Yaskawa INFORM job: X2_50&56A(90,0).JBI

/JOB
//NAME X2_50&56A(90,0)
//POS
///NPOS 396,396,396,18,0,0
///TOOL 0
///POSTYPE PULSE
///PULSE
C00000=35013,-75230,-81678,29902,96544,-59223
C00001=35013,-75230,-81678,29902,96544,50582
C00002=120856,-140422,-87858,-20775,49685,84873
C00003=94802,-63197,-51322,-24283,84063,77554
C00004=130027,34169,-1600,32218,111617,-60978
C00005=146238,55672,63206,30358,82483,-64229
C00006=147931,55156,65583,30589,80380,-64138
C00007=88821,-39952,-28103,-20433,93116,74064
C00008=88821,-39522,-26790,-20414,92564,74158
C00009=88821,-39864,-27834,-20427,93002,74084
C00010=88103,-42626,-29535,-20492,92474,73914
C00011=88821,-39864,-27834,-20427,93002,74084
C00012=78489,-20820,-14449,-12623,103903,88788
C00013=79217,-21691,-15077,-12445,103957,89045
C00014=78489,-21142,-15590,-12658,104428,88732
C00015=86357,-31648,-34432,-18066,105893,79829
C00016=106408,-49809,-40215,-13540,104251,87431
C00017=105408,-58256,-44905,-13671,102667,87249
C00018=105408,-58256,-44905,-13671,102667,87249
C00019=110503,10444,25613,-12126,95572,-74078
C00020=112000,-36737,-25207,-22040,88152,-84766
C00021=112000,-31881,-11932,-22145,82876,-83796
C00022=112000,-30399,-8347,-22203,81533,-83546
C00023=112000,-31881,-11932,-22145,82876,-83796
C00024=116556,-31988,-11028,-21876,83512,-82269
C00025=116556,-30496,-7483,-21927,82195,-82028
C00026=116476,-32903,-9067,-21944,81929,-82006
C00027=116556,-30496,-7483,-21927,82195,-82028
C00028=116556,-30496,-7483,-21927,82195,-82028
C00029=115731,-30414,-7427,-21987,81986,-82285
C00030=116556,-30496,-7483,-21927,82195,-82028
C00031=106621,-34317,-21280,-11409,87224,-86882
C00032=68546,9416,10683,-17932,104217,-63227
C00033=68516,6763,11888,-17759,102202,-62934
C00034=69948,4612,13298,-17270,100624,-62182
C00035=69948,5621,16125,-17192,99456,-62015
C00036=69948,5087,14650,-17232,100063,-62102
C00037=67463,10522,20606,-17770,98699,-62796
C00038=66929,8958,19215,-17898,98632,-62977
C00039=67463,10522,20606,-17770,98699,-62796
C00040=68831,9536,19728,-17449,99024,-62352
C00041=69409,8421,18742,-17312,99180,-62168
C00042=68137,9624,17362,-17710,100309,-62790
C00043=69946,10003,12499,-17525,103743,-62639
C00044=115698,-30544,-51433,-15731,84190,-63390
C00045=118338,-32636,-46922,-7735,73478,-10834
C00046=113479,46792,28572,-8285,94763,37933
C00047=101095,55404,42650,-8147,89306,34054
C00048=100229,58556,52121,-8145,85049,34033
C00049=99767,59813,55030,-8149,83870,33952
C00050=99764,60521,57124,-8160,82954,34012
C00051=99767,59813,55030,-8149,83870,33952
C00052=102778,57366,53086,-13194,83019,35153
C00053=102079,58061,53874,-13178,82781,34934
C00054=102778,57366,53086,-13194,83019,35153
C00055=103317,56175,50346,-13188,84155,35220
C00056=104672,52489,39292,-13191,89159,35160
C00057=104701,56902,48819,-15320,94256,69233
C00058=104701,57353,50315,-15300,93589,69317
C00059=104701,57270,50045,-15303,93709,69302
C00060=104511,53820,46175,-15336,94260,69166
C00061=104638,55892,48016,-15323,94215,69218
C00062=105717,54144,46059,-15234,94714,69537
C00063=105635,50040,42095,-15252,95019,69470
C00064=105236,50331,42415,-15286,94898,69344
C00065=105635,49167,38717,-15311,96595,69274
C00066=102055,-19938,-28050,-3892,79498,23263
C00067=101482,-35884,-39735,-11033,71484,5125
C00068=99031,-31158,-27485,-14483,64579,4851
C00069=99281,-29511,-26374,-14550,64779,4920
C00070=99247,-29735,-26526,-14541,64752,4910
C00071=99247,-29464,-25406,-14605,64218,4980
C00072=99051,-31169,-27981,-14456,64871,4820
C00073=96268,-39480,-34083,-4840,61268,-4619
C00074=96136,-35876,-28725,-4851,59820,-4606
C00075=95241,-35325,-28368,-4481,59831,-4954
C00076=96136,-35958,-29023,-4844,59961,-4612
C00077=124050,-15750,-20412,-8746,80746,42462
C00078=136003,-35750,-34405,-10595,80538,46616
C00079=134863,-34094,-26254,-10570,76291,46583
C00080=136016,-32722,-22756,-10798,75019,47102
C00081=136016,-31890,-20154,-10854,73866,47205
C00082=136016,-32408,-21756,-10817,74572,47142
C00083=116377,-35025,-23683,16914,73563,39729
C00084=116394,-34210,-21577,16985,72720,39615
C00085=115269,-34083,-21492,17148,72970,39239
C00086=117663,-35285,-24614,16688,73723,40220
C00087=141315,-33561,-31051,-11181,80302,48491
C00088=136363,-34899,-19347,-7835,84694,46414
C00089=120104,-33911,-11600,-8301,78857,41249
C00090=118071,-31578,-6204,-8386,76551,40710
C00091=117257,-30555,-3964,-8424,75624,40496
C00092=117257,-29687,-2023,-8450,74882,40547
C00093=117257,-30555,-3964,-8424,75624,40496
C00094=122539,-29708,-1883,-13613,75634,42844
C00095=121317,-29732,-1900,-13643,75432,42443
C00096=122539,-29708,-1883,-13613,75634,42844
C00097=123471,-30618,-3978,-13546,76585,43059
C00098=125796,-32661,-9010,-13387,78955,43601
C00099=120122,-41338,-8990,-8476,73493,41622
C00100=117871,-38446,-3197,-8601,71207,41016
C00101=116972,-37197,-791,-8654,70286,40775
C00102=116972,-36136,1298,-8692,69554,40829
C00103=116972,-37197,-791,-8654,70286,40775
C00104=122649,-36403,912,-13956,70634,43458
C00105=121298,-36427,896,-13995,70410,43017
C00106=122649,-36403,912,-13956,70634,43458
C00107=120043,-14467,15179,-12402,85308,69300
C00108=120029,-16401,14941,-12417,84477,69377
C00109=120021,-18007,13765,-12421,84376,69384
C00110=120029,-16401,14941,-12417,84477,69377
C00111=123681,-37514,-1336,-13860,71590,43701
C00112=126252,-40055,-6735,-13636,73968,44314
C00113=154326,-120554,-77654,-11334,79888,63138
C00114=167720,-105639,-119673,-16034,110248,69380
C00115=180425,17295,-38776,-18903,121217,77748
C00116=161552,-71669,-79142,-10296,105844,81662
C00117=160864,-75997,-77577,-10180,102620,81695
C00118=159718,-74822,-75193,-10227,101627,81377
C00119=159595,-74270,-73499,-10203,100862,81396
C00120=160050,-75992,-74945,-10170,100925,81551
C00121=160240,-80173,-76229,-10103,99611,81726
C00122=160318,-76812,-75188,-10139,100690,81664
C00123=161300,-71121,-77557,-10275,105130,81635
C00124=122590,-90956,-95479,6285,107811,74232
C00125=122432,-96187,-93928,6136,104200,73988
C00126=122366,-98076,-93201,6086,102795,73894
C00127=122349,-96392,-90986,6070,102302,73864
C00128=122333,-96702,-91360,6071,102373,73862
C00129=121172,-100063,-92157,5915,101229,73400
C00130=122333,-96702,-91360,6071,102373,73862
C00131=116908,-96303,-91435,5489,103011,71994
C00132=118888,-98383,-91954,5688,102128,72646
C00133=116908,-96303,-91435,5489,103011,71994
C00134=117392,-89431,-93773,5700,107925,72394
C00135=123779,-92334,-96085,-11860,100478,68930
C00136=121799,-96099,-93963,-11739,97018,68578
C00137=120978,-97397,-93019,-11702,95677,68421
C00138=120976,-95732,-90808,-11689,95182,68467
C00139=121047,-96000,-91535,-11697,95495,68462
C00140=119860,-99344,-92335,-11668,94123,68181
C00141=121047,-96000,-91535,-11697,95495,68462
C00142=119543,-98346,-92112,-11677,94445,68041
C00143=121592,-100306,-92571,-11657,94029,68789
C00144=119543,-98346,-92112,-11677,94445,68041
C00145=122418,-93690,-95360,-11815,99162,68586
C00146=124052,-92327,-98574,-11935,102020,68874
C00147=122075,-96496,-96608,-11789,98453,68536
C00148=121256,-97943,-95721,-11744,97072,68385
C00149=121250,-96320,-93531,-11728,96567,68431
C00150=121163,-96877,-94234,-11732,96698,68388
C00151=119974,-100369,-95083,-11696,95280,68111
C00152=121163,-96877,-94234,-11732,96698,68388
C00153=120506,-98881,-94746,-11711,95903,68236
C00154=118500,-96784,-94222,-11730,96355,67499
C00155=120506,-98881,-94746,-11711,95903,68236
C00156=123349,-93657,-97773,-11879,100767,68753
C00157=136369,-86264,-75827,-53025,86694,81775
C00158=132228,-88122,-74116,-52932,83075,81639
C00159=130522,-88702,-73354,-52914,81621,81560
C00160=129603,-91514,-73993,-52982,80442,81751
C00161=133099,-92681,-76573,-53031,83062,82125
C00162=131615,-95137,-76568,-53090,81428,82278
C00163=130003,-92998,-74814,-53028,80513,81930
C00164=131615,-95137,-76568,-53090,81428,82278
C00165=125724,-93998,-78752,-52538,79248,80319
C00166=127169,-93644,-77288,-52734,79625,80891
C00167=125724,-93998,-78752,-52538,79248,80319
C00168=131917,-91951,-81421,-52749,84465,80650
C00169=125882,-96985,-97972,-20817,92084,56602
C00170=122325,-98161,-95172,-20440,89016,55857
C00171=120880,-94284,-92066,-20293,88735,55390
C00172=120880,-94153,-90803,-20292,88068,55501
C00173=120880,-94284,-92066,-20293,88735,55390
C00174=119026,-94251,-92054,-20095,88291,54803
C00175=120880,-94284,-92066,-20293,88735,55390
C00176=120884,-98206,-92897,-20294,87320,55628
C00177=120880,-94284,-92066,-20293,88735,55390
C00178=125854,-95536,-95978,-20803,91624,56671
C00179=125850,-66912,-79659,-30836,57983,58657
C00180=122561,-63207,-75462,-29110,56252,57732
C00181=121295,-61670,-73737,-28426,55590,57365
C00182=121291,-60661,-71640,-28674,54906,57565
C00183=121285,-60765,-71809,-28654,54949,57550
C00184=119473,-60737,-71796,-27523,54360,56906
C00185=121285,-60765,-71809,-28654,54949,57550
C00186=119935,-60692,-71734,-27818,54496,57075
C00187=119959,-57359,-70502,-27528,55354,56840
C00188=119935,-60692,-71734,-27818,54496,57075
C00189=124401,-66105,-77764,-30230,56821,58377
C00190=128142,-64639,-90036,-18676,74706,62694
C00191=138485,-71827,-101197,11106,105399,77644
C00192=147024,-87385,-83593,35439,109592,87133
C00193=149732,-92665,-83137,35225,106008,87097
C00194=151109,-95679,-83834,35232,104517,87192
C00195=150643,-92710,-80195,35037,104118,86860
C00196=144971,-96193,-77741,39215,100748,74661
C00197=143884,-94649,-78323,39224,102144,74704
C00198=141496,-90316,-79520,39399,105550,74933
C00199=154875,-73459,-94031,-3699,115712,75473
C00200=154642,-88430,-80864,-46638,100530,71967
C00201=150685,-92332,-80273,-46535,96810,71811
C00202=149068,-93915,-80023,-46523,95290,71747
C00203=152233,-91403,-76041,-46197,96115,72893
C00204=138023,-100193,-87798,-32403,89280,71025
C00205=139486,-99224,-88637,-32451,90704,71199
C00206=143008,-96307,-90518,-32622,94313,71562
C00207=126401,-92982,-99947,-26116,71912,46119
C00208=122401,-89174,-95921,-24616,70248,44972
C00209=121170,-87691,-94393,-24143,69731,44617
C00210=121073,-40431,-77118,-23973,104037,41292
C00211=121948,-141376,-105315,-24084,72465,47862
C00212=119793,-124223,-100539,-21665,86903,40754
C00213=121070,-126388,-102412,-21638,87354,41108
C00214=126026,-127807,-105919,-21532,89991,42436
C00215=136654,-67846,-101646,5444,103045,74682
C00216=128322,-96725,-99076,-14451,99613,67284
C00217=128011,-95143,-96681,-14417,98917,67259
C00218=125059,-98267,-95078,-14269,95825,66574
C00219=132883,-103944,-96240,-14189,95056,69399
C00220=122114,-97273,-96139,-7492,99903,69823
C00221=123656,-92823,-98050,-7552,103478,70135
C00222=148370,-106244,-91268,-32547,97235,62203
C00223=143957,-109023,-89633,-32719,93465,61524
C00224=142187,-110300,-89017,-32799,91899,61269
C00225=110014,-102343,-95219,-10833,94604,66470
C00226=122878,-112804,-97097,-10537,93258,71032
C00227=110561,-104342,-93907,-1603,99479,78541
C00228=110841,-84726,-85708,-1760,111290,78449
C00229=111201,-78802,-86432,-1737,114786,78527
C00230=107617,-60482,-79878,-8180,107350,64339
C00231=106036,-64346,-78204,-8057,104211,64009
C00232=105256,-65205,-77316,-8026,103160,63809
C00233=107559,-69233,-78771,-7955,102216,64664
C00234=165613,-100062,-83585,-4761,94184,85074
C00235=168997,-99278,-82863,-4484,94340,86226
C00236=170567,-98725,-82495,-4354,94483,86758
C00237=166939,-94886,-91891,-4771,102005,85231
C00238=180121,-120623,-113011,-11864,94268,89792
C00239=202989,-63880,-99903,-47799,99542,84030
C00240=168472,-147890,-132681,-14947,97151,71352
C00241=154326,-120554,-77654,-11334,79888,63138
C00242=128098,-77833,-51544,1657,63239,16727
C00243=116532,-49017,-34945,4360,90951,81305
C00244=116532,-49017,-34945,4360,90951,81305
C00245=116798,-50663,-32111,4378,88355,81305
C00246=118979,-64696,-37015,4666,76602,81617
C00247=127924,-64268,-36804,4494,76190,84659
C00248=124228,-50732,-32149,5002,87911,83800
C00249=145745,-14259,570,-10366,107018,74117
C00250=151803,-16835,2182,-12669,103763,71943
C00251=152120,-15652,4819,-12499,102817,72155
C00252=153130,-16591,-3293,-13485,106909,71001
C00253=99208,-22167,-7317,16130,105202,90552
C00254=102975,-22456,-1750,16076,101623,90323
C00255=102764,-21603,-119,15971,101119,90180
C00256=102764,-21410,336,15959,100945,90157
C00257=100868,-20755,-6903,14931,106373,89315
C00258=123764,-49143,-35016,4968,90511,83746
C00259=123498,-46334,-32145,-14225,106729,81506
C00260=122671,-49917,-31274,-14287,104276,81501
C00261=124642,-51419,-28814,-13533,102390,82429
C00262=121239,-51674,-29154,-14566,101882,81278
C00263=121239,-51674,-29154,-14566,101882,81278
C00264=121239,-51674,-29154,-14566,101882,81278
C00265=119414,-50002,-31488,-15265,103772,80384
C00266=116044,-49795,-31370,-16241,103155,79243
C00267=108003,-52785,-29324,-8850,97765,81124
C00268=118660,-64605,-35307,-15810,90578,70895
C00269=127566,-70492,-45301,-19994,92283,73343
C00270=120368,-46468,-32388,-15179,106240,80415
C00271=103583,-18395,-21065,-18333,98049,47386
C00272=95522,-2033,346,-19157,86542,33647
C00273=95065,-1179,4289,-19188,84551,33796
C00274=94955,-858,5669,-19196,83900,33869
C00275=92999,-12490,-3621,-19193,83196,33279
C00276=91633,5412,10982,-17435,91860,45178
C00277=96102,40486,49560,-22978,105705,40202
C00278=95175,38955,47637,-23356,105815,39825
C00279=95175,41860,54365,-23036,103374,40320
C00280=96604,40287,46680,-23025,107388,40051
C00281=97434,43818,44752,-23189,110389,39758
C00282=95302,21282,15864,-17128,100326,40606
C00283=95633,-1961,-1285,-16168,78923,31701
C00284=94125,315,3726,-16087,76781,31446
C00285=94086,2267,8889,-16221,74681,31714
C00286=93769,3603,11937,-16272,73472,31765
C00287=95210,13761,20912,-16469,73473,32289
C00288=95827,11154,15194,-16384,75690,32206
C00289=95302,10808,12912,-16245,76762,31872
C00290=94760,268,4885,-16208,76196,31753
C00291=94118,1970,8158,-16204,74972,31685
C00292=93771,3565,12382,-16293,73191,31803
C00293=95246,13304,20868,-16485,73277,32327
C00294=95842,10702,14076,-16353,76128,32151
C00295=96013,9170,10401,-16290,77582,32017
C00296=97216,11756,13085,-16445,77515,32459
C00297=97106,13151,16539,-16517,76140,32606
C00298=96699,14660,19946,-16558,74788,32646
C00299=97321,19796,24727,-16651,74625,32895
C00300=91528,6104,12814,-7587,65442,17765
C00301=89231,-9641,862,-3829,57239,21101
C00302=86569,-23656,-15616,-815,55978,22098
C00303=99387,-43194,-40222,-6284,61646,26942
C00304=121163,28995,9538,-19255,89803,33709
C00305=111536,74157,50908,-19383,94154,29578
C00306=110126,77328,60869,-19265,89563,29800
C00307=109597,77904,61840,-18115,89315,29667
C00308=107134,62574,43702,-13173,82287,21832
C00309=105849,37660,21975,-10686,72529,22941
C00310=108144,30390,14425,-11303,73735,23647
C00311=110038,48233,28322,-17563,85893,26316
C00312=110492,45790,38116,-18907,91301,38258
C00313=109482,39772,34705,-18931,90124,38079
C00314=108901,41209,40132,-18939,87523,38277
C00315=108525,40703,40973,-18962,86700,38272
C00316=107041,55931,58526,-17360,94880,40074
C00317=107089,67852,69975,-15460,97104,40498
C00318=107063,68178,67130,-13775,98442,40242
C00319=113418,36081,17598,-23566,90539,39080
C00320=113418,36081,17598,-23168,95829,82784
C00321=113828,51923,41074,-24171,98232,82423
C00322=112579,52431,41633,-24296,97790,82045
C00323=112126,56349,44369,-24366,97957,81836
C00324=108217,58430,46714,-24702,96454,80681
C00325=108494,54192,43684,-24661,96249,80828
C00326=108007,54490,44017,-24701,96056,80686
C00327=107594,60273,47410,-24788,96737,80387
C00328=114507,54753,41023,-24220,99790,82353
C00329=122054,71046,63948,-32664,112221,61348
C00330=123579,46190,40204,-38346,104555,54529
C00331=124736,37096,33930,-39238,101677,53630
C00332=124818,38918,39542,-38856,99735,54394
C00333=126462,40069,35828,-39705,101719,52991
C00334=128176,30389,18653,-40526,106846,51750
C00335=130467,-19777,-28453,-43779,86857,-28489
C00336=121945,-40313,-29836,-49261,62361,-22447
C00337=123791,-37570,-24592,-50353,62174,-21277
C00338=114538,-37294,-24521,-48212,57212,-23703
C00339=116456,-42529,-32983,-47605,59952,-24171
C00340=113288,-38496,-19602,-52049,50370,-20126
C00341=111978,-38266,-19460,-51659,49655,-20498
C00342=111880,-40713,-23013,-51024,50195,-20951
C00343=122010,-41537,-23518,-53640,55853,-18263
C00344=118733,-42874,-23495,-50076,50608,-22105
C00345=115692,-42672,-23415,-49110,48994,-23003
C00346=119979,-48793,-33564,-48599,53387,-23123
C00347=127641,-44516,-39522,-49206,67999,-22470
C00348=137272,-90960,-86846,-29989,75596,51153
C00349=137772,-94948,-88443,-30238,74846,51554
C00350=80124,-23753,-1605,24425,88616,-57626
C00351=97606,38320,19913,32229,69524,-73177
C00352=104908,49911,44038,31966,59160,-73213
C00353=105731,66374,62732,32681,56250,-73801
C00354=101009,56188,45401,32602,62685,-73830
C00355=95324,41633,28025,33647,67650,-74589
C00356=87558,19072,373,28757,109210,-81139
C00357=99257,11218,8118,26405,109034,-79116
C00358=100705,8698,11538,26232,105511,-79373
C00359=103992,6523,9295,19718,103157,-78424
C00360=103706,6801,9674,20068,103243,-78529
C00361=103706,6801,9674,20068,103243,-78529
C00362=103175,12796,9745,21520,108066,-80350
C00363=94457,17964,8722,13249,111502,-83272
C00364=77268,-3254,-24039,37164,82398,-77433
C00365=55933,-99496,-79908,41589,80337,-87481
C00366=92475,-142040,-80472,-3538,45591,39607
C00367=111759,-138997,-77779,-20724,42469,82604
C00368=123409,-124840,-68778,-23994,47004,86899
C00369=115111,-123372,-67292,-17121,44583,82853
C00370=106159,-121342,-66429,-9144,43886,78109
C00371=56877,-95499,-59936,14598,58195,57192
C00372=67543,-97387,-64583,11943,58838,61427
C00373=85335,-36233,-33573,-15386,101650,67363
C00374=22776,-147712,-91578,22852,59519,43831
C00375=66236,-86626,-72800,11302,69406,62015
C00376=122101,-60707,-49124,40437,82186,-58582
C00377=76878,-31978,-23741,-7994,99594,69431
C00378=79357,-35161,-25830,-10416,97591,64533
C00379=82324,-46618,-32975,-14804,90128,52114
C00380=86643,-46469,-34772,-14478,92051,53396
C00381=73286,-4461,-1127,-6755,115907,88976
C00382=73225,-6334,-1269,-6726,115035,89004
C00383=71733,-2264,5245,-7236,112998,88564
C00384=76479,-5255,-4471,-10939,116481,85182
C00385=98335,-62985,-54253,-3239,96100,60563
C00386=98335,-62985,-54253,-3239,96100,60563
C00387=98335,-62985,-54253,-3239,96100,60563
C00388=152493,16707,-760,-6447,101329,44907
C00389=169300,37694,50213,-44743,100506,44736
C00390=167112,29738,44456,-45250,99025,44384
C00391=162955,52490,68578,-45996,94710,44438
C00392=158969,29363,17393,-36895,102134,39004
C00393=132653,-84295,-81500,4027,86761,-71858
C00394=118286,-84176,-81449,4028,86790,-71859
C00395=-2286,-108146,-98365,80,72600,-100
BC00000=231000,517456,593434
BC00001=34376,517456,225147
BC00002=102572,425363,301105
BC00003=102572,425363,301105
BC00004=334489,491452,488918
BC00005=322698,517456,378589
BC00006=322698,517456,378589
BC00007=102572,425363,301105
BC00008=102572,425363,301105
BC00009=102572,425363,301105
BC00010=102572,425363,301105
BC00011=102572,425363,301105
BC00012=102572,425363,301105
BC00013=102572,425363,301105
BC00014=102572,425363,301105
BC00015=102572,425363,301105
BC00016=102572,425363,301105
BC00017=102572,579800,381307
BC00018=306896,476295,640078
BC00019=306896,448601,572655
BC00020=271432,459376,401351
BC00021=271432,459376,401351
BC00022=271432,459376,401351
BC00023=271432,459376,401351
BC00024=271432,459376,401351
BC00025=271432,459376,401351
BC00026=271432,459376,401351
BC00027=271432,459376,401351
BC00028=271432,459376,401351
BC00029=271432,459376,401351
BC00030=271432,459376,401351
BC00031=271432,459376,401351
BC00032=268738,434477,371771
BC00033=268738,434477,371771
BC00034=268738,434477,371771
BC00035=268738,434477,371771
BC00036=268738,434477,371771
BC00037=268738,434477,371771
BC00038=268738,434477,371771
BC00039=268738,434477,371771
BC00040=268738,434477,371771
BC00041=268738,434477,371771
BC00042=268738,434477,371771
BC00043=268738,434477,371771
BC00044=294080,442709,254978
BC00045=331538,416726,228027
BC00046=305027,399020,290854
BC00047=305027,399020,290854
BC00048=305027,399020,290854
BC00049=305027,399020,290854
BC00050=305027,399020,290854
BC00051=305027,399020,290854
BC00052=305027,399020,290854
BC00053=305027,399020,290854
BC00054=305027,399020,290854
BC00055=305027,399020,290854
BC00056=305027,399020,290854
BC00057=305029,399021,290852
BC00058=305029,399021,290852
BC00059=305029,399021,290852
BC00060=305029,399021,290852
BC00061=305029,399021,290852
BC00062=305029,399021,290852
BC00063=305029,399021,290852
BC00064=305029,399021,290852
BC00065=305029,399021,290852
BC00066=305029,399021,290852
BC00067=305029,399021,290852
BC00068=305029,399021,290852
BC00069=305029,399021,290852
BC00070=305029,399021,290852
BC00071=305029,399021,290852
BC00072=305029,399021,290852
BC00073=305029,399021,290852
BC00074=305029,399021,290852
BC00075=305029,399021,290852
BC00076=305029,399021,290852
BC00077=334039,399020,360133
BC00078=334039,399020,360133
BC00079=334039,399020,360133
BC00080=334039,399020,360133
BC00081=334039,399020,360133
BC00082=334039,399020,360133
BC00083=334039,399020,360133
BC00084=334039,399020,360133
BC00085=334039,399020,360133
BC00086=334039,399020,360133
BC00087=334039,399020,360133
BC00088=367859,399020,440892
BC00089=367859,399020,440892
BC00090=367859,399020,440892
BC00091=367859,399020,440892
BC00092=367859,399020,440892
BC00093=367859,399020,440892
BC00094=367859,399020,440892
BC00095=367859,399020,440892
BC00096=367859,399020,440892
BC00097=367859,399020,440892
BC00098=367859,399020,440892
BC00099=367957,451741,487073
BC00100=367957,451741,487073
BC00101=367957,451741,487073
BC00102=367957,451741,487073
BC00103=367957,451741,487073
BC00104=367957,451741,487073
BC00105=367957,451741,487073
BC00106=367957,451741,487073
BC00107=367957,451741,487073
BC00108=367957,451741,487073
BC00109=367957,451741,487073
BC00110=367957,451741,487073
BC00111=367957,451741,487073
BC00112=367957,451741,487073
BC00113=242061,521422,834580
BC00114=140834,449782,1062640
BC00115=97513,455583,1075193
BC00116=1592,411167,1075139
BC00117=1592,411167,1075139
BC00118=1592,409938,1075139
BC00119=1592,409938,1075139
BC00120=1592,409938,1075139
BC00121=1592,409938,1075139
BC00122=1592,409938,1075139
BC00123=1592,409938,1075139
BC00124=50980,356914,1075139
BC00125=50980,356914,1075139
BC00126=50980,356914,1075139
BC00127=50980,356914,1075139
BC00128=50980,356914,1075139
BC00129=50980,356914,1075139
BC00130=50980,356914,1075139
BC00131=50980,356914,1075139
BC00132=50980,356914,1075139
BC00133=50980,356914,1075139
BC00134=50980,356914,1075139
BC00135=20406,370413,1075139
BC00136=20406,370413,1075139
BC00137=20406,370413,1075139
BC00138=20406,370413,1075139
BC00139=20406,370413,1075139
BC00140=20406,370413,1075139
BC00141=20406,370413,1075139
BC00142=20406,370413,1075139
BC00143=20406,370413,1075139
BC00144=20406,370413,1075139
BC00145=20406,370413,1075139
BC00146=44109,357401,1075139
BC00147=44109,357401,1075139
BC00148=44109,357401,1075139
BC00149=44109,357401,1075139
BC00150=44109,357401,1075139
BC00151=44109,357401,1075139
BC00152=44109,357401,1075139
BC00153=44109,357401,1075139
BC00154=44109,357401,1075139
BC00155=44109,357401,1075139
BC00156=44109,357401,1075139
BC00157=1592,378501,1075139
BC00158=1592,378501,1075139
BC00159=1592,378501,1075139
BC00160=1592,378501,1075139
BC00161=1592,378501,1075139
BC00162=1592,378501,1075139
BC00163=1592,378501,1075139
BC00164=1592,378501,1075139
BC00165=1592,378501,1075139
BC00166=1592,378501,1075139
BC00167=1592,378501,1075139
BC00168=1592,378501,1075139
BC00169=34924,366834,1075139
BC00170=34924,366834,1075139
BC00171=34924,366834,1075139
BC00172=34924,366834,1075139
BC00173=34924,366834,1075139
BC00174=34924,366834,1075139
BC00175=34924,366834,1075139
BC00176=34924,366834,1075139
BC00177=34924,366834,1075139
BC00178=34924,366834,1075139
BC00179=29635,379683,1075139
BC00180=29635,379683,1075139
BC00181=29635,379683,1075139
BC00182=29635,379683,1075139
BC00183=29635,379683,1075139
BC00184=29635,379683,1075139
BC00185=29635,379683,1075139
BC00186=29635,379683,1075139
BC00187=29635,379683,1075139
BC00188=29635,379683,1075139
BC00189=29635,379683,1075139
BC00190=45948,369971,1075139
BC00191=91010,343142,1075139
BC00192=128368,320900,1075139
BC00193=128368,320900,1075139
BC00194=128368,320900,1075139
BC00195=128368,320900,1075139
BC00196=128368,320900,1075139
BC00197=128368,320900,1075139
BC00198=128368,320900,1075139
BC00199=82932,344066,1075139
BC00200=34742,368635,1075139
BC00201=34742,368635,1075139
BC00202=34742,368635,1075139
BC00203=34742,368635,1075139
BC00204=34742,368635,1075139
BC00205=34742,368635,1075139
BC00206=34742,368635,1075139
BC00207=32385,335579,1075139
BC00208=32385,335579,1075139
BC00209=32385,335579,1075139
BC00210=32385,335579,1075139
BC00211=32385,335579,1075139
BC00212=32385,335579,1075139
BC00213=32385,335579,1075139
BC00214=32385,335579,1075139
BC00215=83004,347908,1075139
BC00216=56012,350823,1075139
BC00217=56012,350823,1075139
BC00218=56012,350822,1075135
BC00219=56012,350822,1075135
BC00220=56012,350823,1075139
BC00221=56012,350823,1075139
BC00222=32229,352573,1075139
BC00223=32229,352573,1075139
BC00224=32229,352573,1075139
BC00225=32229,352573,1075139
BC00226=32229,352573,1075139
BC00227=32229,352573,1075139
BC00228=32229,352573,1075139
BC00229=32229,352573,1075139
BC00230=1592,390224,1075139
BC00231=1592,390224,1075139
BC00232=1592,390224,1075139
BC00233=1592,390224,1075139
BC00234=1592,390224,1075139
BC00235=1592,390224,1075139
BC00236=1592,390224,1075139
BC00237=1592,390224,1075139
BC00238=1592,390224,1075139
BC00239=97513,454354,1075193
BC00240=140834,448553,1062640
BC00241=242061,520193,834580
BC00242=311361,456270,477376
BC00243=342823,443238,375594
BC00244=342823,443238,375594
BC00245=342823,443238,375594
BC00246=342823,443238,375594
BC00247=342823,443238,375594
BC00248=342823,443238,375594
BC00249=342823,443238,375594
BC00250=342823,443238,375594
BC00251=342823,443238,375594
BC00252=342823,443238,375594
BC00253=342823,443238,375594
BC00254=342823,443238,375594
BC00255=342823,443238,375594
BC00256=342823,443238,375594
BC00257=342823,443238,375594
BC00258=342823,443238,375594
BC00259=362743,414004,329031
BC00260=362743,414004,329031
BC00261=362743,414004,329031
BC00262=362743,414004,329031
BC00263=362743,414004,329031
BC00264=362743,414004,329031
BC00265=362743,414004,329031
BC00266=362743,414004,329031
BC00267=362743,414004,329031
BC00268=362743,414004,329031
BC00269=362743,414004,329031
BC00270=362743,414004,329031
BC00271=315566,460561,335729
BC00272=294603,481248,338705
BC00273=294603,481248,338705
BC00274=294603,481247,338705
BC00275=294603,481247,338705
BC00276=294603,481247,338705
BC00277=294603,481248,338705
BC00278=294603,481248,338705
BC00279=294603,481248,338705
BC00280=294603,481248,338705
BC00281=294603,481248,338705
BC00282=294603,481248,338705
BC00283=290459,488683,355824
BC00284=290459,488683,355824
BC00285=290459,488683,355824
BC00286=290459,488683,355824
BC00287=290459,488683,355824
BC00288=290459,488683,355824
BC00289=290459,488683,355824
BC00290=290354,460436,354488
BC00291=290354,460436,354488
BC00292=290354,460436,354488
BC00293=290354,460436,354488
BC00294=290354,460436,354488
BC00295=290354,460436,354488
BC00296=293273,446294,341840
BC00297=293273,446294,341840
BC00298=293273,446294,341840
BC00299=293273,446294,341840
BC00300=293273,446294,341840
BC00301=293273,446294,341840
BC00302=293273,446294,341840
BC00303=293273,446294,341840
BC00304=316572,397791,307269
BC00305=317775,402370,174220
BC00306=317775,402370,174220
BC00307=317775,402370,174220
BC00308=317775,402370,174220
BC00309=317775,402370,219932
BC00310=317775,402370,258168
BC00311=317775,402370,227987
BC00312=319614,400694,306223
BC00313=319614,400694,306223
BC00314=319614,400694,306223
BC00315=319614,400694,306223
BC00316=319614,400694,306223
BC00317=319614,400694,306223
BC00318=319614,400694,306223
BC00319=319614,400694,252456
BC00320=319614,400694,252456
BC00321=319614,400694,252456
BC00322=319614,400694,252456
BC00323=319614,400694,252456
BC00324=319614,400694,252456
BC00325=319614,400694,252456
BC00326=319614,400694,252456
BC00327=319614,400694,252456
BC00328=319614,400694,252456
BC00329=319614,400694,252456
BC00330=319614,400694,252456
BC00331=319610,400694,252455
BC00332=319610,400694,252455
BC00333=319614,400694,252456
BC00334=319614,400694,252456
BC00335=319614,400694,252456
BC00336=319614,400694,252456
BC00337=319614,400694,252456
BC00338=319614,400694,252456
BC00339=319614,400694,252456
BC00340=319614,400694,252456
BC00341=319614,400694,252456
BC00342=319614,400694,252456
BC00343=319614,400694,252456
BC00344=319614,400694,252456
BC00345=319614,400694,252456
BC00346=319614,400694,252456
BC00347=319614,400694,252456
BC00348=319614,400694,392080
BC00349=319614,552522,392080
BC00350=396313,516601,467973
BC00351=396313,490351,238820
BC00352=396313,490351,238820
BC00353=396313,490351,238820
BC00354=396313,490351,238820
BC00355=395126,490351,305637
BC00356=395126,490351,305637
BC00357=395126,490351,305637
BC00358=395126,490351,305637
BC00359=395126,490351,305637
BC00360=395126,490351,305637
BC00361=395126,490351,305637
BC00362=395126,490351,305637
BC00363=395126,490351,305637
BC00364=391357,490351,517866
BC00365=391357,520423,517866
BC00366=172219,466569,359308
BC00367=102572,425363,301105
BC00368=102572,425363,301105
BC00369=97784,424339,294147
BC00370=102572,425363,301105
BC00371=102572,425363,301105
BC00372=102572,425363,301105
BC00373=102572,425363,301105
BC00374=102572,425363,301105
BC00375=236824,425363,301105
BC00376=301028,425363,301105
BC00377=102572,425363,301105
BC00378=102572,425363,301105
BC00379=102572,425363,301105
BC00380=102572,425363,301105
BC00381=102572,425363,301105
BC00382=102572,425363,301105
BC00383=102572,425363,301105
BC00384=102572,425363,301105
BC00385=102572,425363,301105
BC00386=102572,544891,301105
BC00387=294297,481237,657653
BC00388=359247,425363,301105
BC00389=359247,425363,301105
BC00390=357450,425363,301105
BC00391=357450,425363,301105
BC00392=357450,425363,301105
BC00393=328822,425363,456749
BC00394=328822,505297,456749
BC00395=84290,517377,1064440
EC00000=-798156,-183832
EC00001=-798156,-183832
EC00002=-798156,-183832
EC00003=-798156,-183832
EC00004=-798156,-183832
EC00005=-798156,-183832
EC00006=-798156,-183832
EC00007=-798156,-183832
EC00008=-798156,-183832
EC00009=-798156,-183832
EC00010=-798156,-183832
EC00011=-798156,-183832
EC00012=-798156,-183832
EC00013=-798156,-183832
EC00014=-798156,-183832
EC00015=-798156,-183832
EC00016=-798156,-183832
EC00017=-798156,-183832
EC00018=-798156,-183832
EC00019=-798156,-183832
EC00020=-798156,-183832
EC00021=-798156,-183832
EC00022=-798156,-183832
EC00023=-798156,-183832
EC00024=-798156,-183832
EC00025=-798156,-183832
EC00026=-798156,-183832
EC00027=-798156,-183832
EC00028=-798156,-183832
EC00029=-798156,-183832
EC00030=-798156,-183832
EC00031=-798156,-183832
EC00032=-798156,-183832
EC00033=-798156,-183832
EC00034=-798156,-183832
EC00035=-798156,-183832
EC00036=-798156,-183832
EC00037=-798156,-183832
EC00038=-798156,-183832
EC00039=-798156,-183832
EC00040=-798156,-183832
EC00041=-798156,-183832
EC00042=-798156,-183832
EC00043=-798156,-183832
EC00044=-798156,-183832
EC00045=-798156,-183832
EC00046=-798156,-183832
EC00047=-798156,-183832
EC00048=-798156,-183832
EC00049=-798156,-183832
EC00050=-798156,-183832
EC00051=-798156,-183832
EC00052=-798156,-183832
EC00053=-798156,-183832
EC00054=-798156,-183832
EC00055=-798156,-183832
EC00056=-798156,-183832
EC00057=-798155,-183832
EC00058=-798155,-183832
EC00059=-798155,-183832
EC00060=-798155,-183832
EC00061=-798155,-183832
EC00062=-798155,-183832
EC00063=-798155,-183832
EC00064=-798155,-183832
EC00065=-798155,-183832
EC00066=-798155,-183832
EC00067=-798155,-183832
EC00068=-798155,-183832
EC00069=-798155,-183832
EC00070=-798155,-183832
EC00071=-798155,-183832
EC00072=-798155,-183832
EC00073=-798155,-183832
EC00074=-798155,-183832
EC00075=-798155,-183832
EC00076=-798155,-183832
EC00077=-798156,-183832
EC00078=-798156,-183832
EC00079=-798156,-183832
EC00080=-798156,-183832
EC00081=-798156,-183832
EC00082=-798156,-183832
EC00083=-798156,-183832
EC00084=-798156,-183832
EC00085=-798156,-183832
EC00086=-798156,-183832
EC00087=-798156,-183832
EC00088=-798156,-183832
EC00089=-798156,-183832
EC00090=-798156,-183832
EC00091=-798156,-183832
EC00092=-798156,-183832
EC00093=-798156,-183832
EC00094=-798156,-183832
EC00095=-798156,-183832
EC00096=-798156,-183832
EC00097=-798156,-183832
EC00098=-798156,-183832
EC00099=-798156,-183832
EC00100=-798156,-183832
EC00101=-798156,-183832
EC00102=-798156,-183832
EC00103=-798156,-183832
EC00104=-798156,-183832
EC00105=-798156,-183832
EC00106=-798156,-183832
EC00107=-798156,-183832
EC00108=-798156,-183832
EC00109=-798156,-183832
EC00110=-798156,-183832
EC00111=-798156,-183832
EC00112=-798156,-183832
EC00113=-860042,-183832
EC00114=-895167,-183832
EC00115=-929003,-183832
EC00116=-975524,-183832
EC00117=-975524,-183832
EC00118=-975524,-183832
EC00119=-975524,-183832
EC00120=-975524,-183832
EC00121=-975524,-183832
EC00122=-975524,-183832
EC00123=-975524,-183832
EC00124=-975524,-183832
EC00125=-975524,-183832
EC00126=-975524,-183832
EC00127=-975524,-183832
EC00128=-975524,-183832
EC00129=-975524,-183832
EC00130=-975524,-183832
EC00131=-975524,-183832
EC00132=-975524,-183832
EC00133=-975524,-183832
EC00134=-975524,-183832
EC00135=-975524,-183832
EC00136=-975524,-183832
EC00137=-975524,-183832
EC00138=-975524,-183832
EC00139=-975524,-183832
EC00140=-975524,-183832
EC00141=-975524,-183832
EC00142=-975524,-183832
EC00143=-975524,-183832
EC00144=-975524,-183832
EC00145=-975524,-183832
EC00146=-975524,-183832
EC00147=-975524,-183832
EC00148=-975524,-183832
EC00149=-975524,-183832
EC00150=-975524,-183832
EC00151=-975524,-183832
EC00152=-975524,-183832
EC00153=-975524,-183832
EC00154=-975524,-183832
EC00155=-975524,-183832
EC00156=-975524,-183832
EC00157=-975524,-183832
EC00158=-975524,-183832
EC00159=-975524,-183832
EC00160=-975524,-183832
EC00161=-975524,-183832
EC00162=-975524,-183832
EC00163=-975524,-183832
EC00164=-975524,-183832
EC00165=-975524,-183832
EC00166=-975524,-183832
EC00167=-975524,-183832
EC00168=-975524,-183832
EC00169=-975524,-183832
EC00170=-975524,-183832
EC00171=-975524,-183832
EC00172=-975524,-183832
EC00173=-975524,-183832
EC00174=-975524,-183832
EC00175=-975524,-183832
EC00176=-975524,-183832
EC00177=-975524,-183832
EC00178=-975524,-183832
EC00179=-975524,-183832
EC00180=-975524,-183832
EC00181=-975524,-183832
EC00182=-975524,-183832
EC00183=-975524,-183832
EC00184=-975524,-183832
EC00185=-975524,-183832
EC00186=-975524,-183832
EC00187=-975524,-183832
EC00188=-975524,-183832
EC00189=-975524,-183832
EC00190=-975524,-183832
EC00191=-975524,-183832
EC00192=-975524,-183832
EC00193=-975524,-183832
EC00194=-975524,-183832
EC00195=-975524,-183832
EC00196=-975524,-183832
EC00197=-975524,-183832
EC00198=-975524,-183832
EC00199=-975524,-183832
EC00200=-975524,-183832
EC00201=-975524,-183832
EC00202=-975524,-183832
EC00203=-975524,-183832
EC00204=-975524,-183832
EC00205=-975524,-183832
EC00206=-975524,-183832
EC00207=-975524,-183832
EC00208=-975524,-183832
EC00209=-975524,-183832
EC00210=-975524,-183832
EC00211=-975524,-183832
EC00212=-975524,-183832
EC00213=-975524,-183832
EC00214=-975524,-183832
EC00215=-975524,-183832
EC00216=-975524,-183832
EC00217=-975524,-183832
EC00218=-975522,-183833
EC00219=-975522,-183833
EC00220=-975524,-183832
EC00221=-975524,-183832
EC00222=-975524,-183832
EC00223=-975524,-183832
EC00224=-975524,-183832
EC00225=-975524,-183832
EC00226=-975524,-183832
EC00227=-975524,-183832
EC00228=-975524,-183832
EC00229=-975524,-183832
EC00230=-975524,-183832
EC00231=-975524,-183832
EC00232=-975524,-183832
EC00233=-975524,-183832
EC00234=-975524,-183832
EC00235=-975524,-183832
EC00236=-975524,-183832
EC00237=-975524,-183832
EC00238=-975524,-183832
EC00239=-929003,-183832
EC00240=-895167,-183832
EC00241=-860042,-183832
EC00242=-817325,-183832
EC00243=-798156,-183832
EC00244=-798156,-183832
EC00245=-798156,-183832
EC00246=-798156,-183832
EC00247=-798156,-183832
EC00248=-798156,-183832
EC00249=-798156,-183832
EC00250=-798156,-183832
EC00251=-798156,-183832
EC00252=-798156,-183832
EC00253=-798156,-183832
EC00254=-798156,-183832
EC00255=-798156,-183832
EC00256=-798156,-183832
EC00257=-798156,-183832
EC00258=-798156,-183832
EC00259=-798156,-183832
EC00260=-798156,-183832
EC00261=-798156,-183832
EC00262=-798156,-183832
EC00263=-798156,-183832
EC00264=-798156,-183832
EC00265=-798156,-183832
EC00266=-798156,-183832
EC00267=-798156,-183832
EC00268=-798156,-183832
EC00269=-798156,-183832
EC00270=-798156,-183832
EC00271=-798156,-183832
EC00272=-798156,-183832
EC00273=-798156,-183832
EC00274=-798154,-183835
EC00275=-798154,-183835
EC00276=-798154,-183835
EC00277=-798156,-183832
EC00278=-798156,-183832
EC00279=-798156,-183832
EC00280=-798156,-183832
EC00281=-798156,-183832
EC00282=-798156,-183832
EC00283=-798156,-183832
EC00284=-798156,-183832
EC00285=-798156,-183832
EC00286=-798156,-183832
EC00287=-798156,-183832
EC00288=-798156,-183832
EC00289=-798156,-183832
EC00290=-798156,-183832
EC00291=-798156,-183832
EC00292=-798156,-183832
EC00293=-798156,-183832
EC00294=-798156,-183832
EC00295=-798156,-183832
EC00296=-798156,-183832
EC00297=-798156,-183832
EC00298=-798156,-183832
EC00299=-798156,-183832
EC00300=-798156,-183832
EC00301=-798156,-183832
EC00302=-798156,-183832
EC00303=-798156,-183832
EC00304=-798156,-183832
EC00305=-798156,-183832
EC00306=-798156,-183832
EC00307=-798156,-183832
EC00308=-798156,-183832
EC00309=-798156,-183832
EC00310=-798156,-183832
EC00311=-798156,-183832
EC00312=-798156,-183832
EC00313=-798156,-183832
EC00314=-798156,-183832
EC00315=-798156,-183832
EC00316=-798156,-183832
EC00317=-798156,-183832
EC00318=-798156,-183832
EC00319=-798156,-183832
EC00320=-798156,-183832
EC00321=-798156,-183832
EC00322=-798156,-183832
EC00323=-798156,-183832
EC00324=-798156,-183832
EC00325=-798156,-183832
EC00326=-798156,-183832
EC00327=-798156,-183832
EC00328=-798156,-183832
EC00329=-798156,-183832
EC00330=-798156,-183832
EC00331=-798155,-183834
EC00332=-798155,-183834
EC00333=-798156,-183832
EC00334=-798156,-183832
EC00335=-798156,-183832
EC00336=-798156,-183832
EC00337=-798156,-183832
EC00338=-798156,-183832
EC00339=-798156,-183832
EC00340=-798156,-183832
EC00341=-798156,-183832
EC00342=-798156,-183832
EC00343=-798156,-183832
EC00344=-798156,-183832
EC00345=-798156,-183832
EC00346=-798156,-183832
EC00347=-798156,-183832
EC00348=-798156,-183832
EC00349=-798156,-183832
EC00350=-798156,-183832
EC00351=-798156,-183832
EC00352=-798156,-183832
EC00353=-798156,-183832
EC00354=-798156,-183832
EC00355=-798156,-183832
EC00356=-798156,-183832
EC00357=-798156,-183832
EC00358=-798156,-183832
EC00359=-798156,-183832
EC00360=-798156,-183832
EC00361=-798156,-183832
EC00362=-798156,-183832
EC00363=-798156,-183832
EC00364=-798156,-183832
EC00365=-798156,-183832
EC00366=-798156,-183832
EC00367=-798156,-183832
EC00368=-798156,-183832
EC00369=-798156,-183832
EC00370=-798156,-183832
EC00371=-798156,-183832
EC00372=-798156,-183832
EC00373=-798156,-183832
EC00374=-798156,-183832
EC00375=-798156,-183832
EC00376=-798156,-183832
EC00377=-798156,-183832
EC00378=-798156,-183832
EC00379=-798156,-183832
EC00380=-798156,-183832
EC00381=-798156,-183832
EC00382=-798156,-183832
EC00383=-798156,-183832
EC00384=-798156,-183832
EC00385=-798156,-183832
EC00386=-798156,-183832
EC00387=-798156,-183832
EC00388=-798156,-183832
EC00389=-798156,-183832
EC00390=-798156,-183832
EC00391=-798156,-183832
EC00392=-798156,-183832
EC00393=-798156,-183832
EC00394=-798156,-183832
EC00395=-798156,-183832
///POSTYPE BASE
///RECTAN
///RCONF 0,0,0,0,1,0,0,0,0,0,0,0,0,0,0,0,0,0,0,0,0,0,0,0
P00006=2.006,1.622,-0.565,0.0000,0.0000,0.0000
P00021=0.073,2.058,-0.109,0.0000,0.0000,0.0000
P00022=2.006,1.622,-0.565,0.0000,0.0000,0.0000
///RCONF 0,0,0,0,0,0,0,0,0,0,0,0,0,0,0,0,0,0,0,0,0,0,0,0
P00023=-2.957,-4.083,2.762,0.0000,0.0000,0.0000
P00024=-1.466,-0.226,-0.419,0.0000,0.0000,0.0000
P00025=3.643,0.007,-2.585,0.0000,0.0000,0.0000
P00026=2.644,0.055,-2.583,0.0000,0.0000,0.0000
P00027=2.278,0.099,-4.210,0.0000,0.0000,0.0000
P00028=-1.778,-0.182,-2.050,0.0000,0.0000,0.0000
P00029=1.749,4.006,-0.261,0.0000,0.0000,0.0000
P00030=-0.014,-0.768,0.131,0.0000,0.0000,0.0000
P00032=-0.423,0.157,3.222,0.0000,0.0000,0.0000
P00033=0.854,-1.099,3.047,0.0000,0.0000,0.0000
///RCONF 0,0,0,0,1,0,0,0,0,0,0,0,0,0,0,0,0,0,0,0,0,0,0,0
P00034=-8.151,9.743,-4.393,0.0000,0.0000,0.0000
///RCONF 0,0,0,0,0,0,0,0,0,0,0,0,0,0,0,0,0,0,0,0,0,0,0,0
P00060=1524.284,698.404,-261.973,-0.4635,36.8346,-1.2388
P00061=1211.499,975.999,-261.374,0.5148,35.2356,175.5099
P00063=1197.217,207.358,-268.729,0.4863,35.2395,175.4586
P00099=-10.497,4.418,3.734,0.0000,0.0000,0.0000
//INST
///DATE 2024/12/09 15:16
///ATTR SC,RW
///GROUP1 RB1,BS1
///GROUP2 ST1
NOP
'X2_50&56A(90,0)
'Down
'Path S3714
SFTOF3D
MOVJ C00000 BC00000 VJ=100.00  +MOVJ EC00000 VJ=100.00
MOVJ C00001 BC00001 VJ=100.00  +MOVJ EC00001 VJ=100.00
MOVJ C00002 BC00002 VJ=100.00  +MOVJ EC00002 VJ=100.00
MOVJ C00003 BC00003 VJ=100.00  +MOVJ EC00003 VJ=100.00
COMM MOVJ C00004 BC00004 VJ=100.00  +MOVJ EC00004 VJ=100.00
COMM MOVJ C00005 BC00005 VJ=100.00  +MOVJ EC00005 VJ=100.00
COMM MOVL C00006 BC00006 V=800.0  +MOVJ EC00006 VJ=100.00
SMOVL C00007 BC00007 V=166.7  +MOVJ EC00007
SREFP 3 C00008 BC00008  +REFP EC00008
CALL JOB:SEARCH-R1-S13D
SET P034 P006
SFTON3D P034
SMOVL C00009 BC00009 V=166.7  +MOVJ EC00009
SREFP 3 C00010 BC00010  +REFP EC00010
CALL JOB:SEARCH-R1-S13D
SET P034 P006
SFTON3D P034
SMOVL C00011 BC00011 V=166.7  +MOVJ EC00011
SMOVL C00012 BC00012 V=166.7  +MOVJ EC00012
SREFP 3 C00013 BC00013  +REFP EC00013
CALL JOB:SEARCH-R1-S13D
SET P034 P006
SFTON3D P034
SMOVL C00014 BC00014 V=133.3  +MOVJ EC00014
SFTOF3D
MOVL C00015 BC00015 V=800.0  +MOVJ EC00015 VJ=100.00
MOVL C00016 BC00016 V=1000.0  +MOVJ EC00016 VJ=100.00
MOVJ C00017 BC00017 VJ=100.00  +MOVJ EC00017 VJ=100.00
MOVJ C00018 BC00018 VJ=100.00  +MOVJ EC00018 VJ=100.00
MOVJ C00019 BC00019 VJ=100.00  +MOVJ EC00019 VJ=100.00
'EndPath S3714
'Path S3715
SFTOF3D
MOVL C00020 BC00020 V=800.0  +MOVJ EC00020 VJ=100.00
SMOVL C00021 BC00021 V=166.7  +MOVJ EC00021
SREFP 3 C00022 BC00022  +REFP EC00022
CALL JOB:SEARCH-R1-S13D
SET P033 P006
SFTON3D P033
SMOVL C00023 BC00023 V=333.3  +MOVJ EC00023
SMOVL C00024 BC00024 V=166.7  +MOVJ EC00024
SMOVL C00025 BC00025 V=166.7  +MOVJ EC00025
SREFP 3 C00026 BC00026  +REFP EC00026
CALL JOB:SEARCH-R1-S13D
SET P033 P006
SFTON3D P033
SMOVL C00027 BC00027 V=166.7  +MOVJ EC00027
SMOVL C00028 BC00028 V=166.7  +MOVJ EC00028
SREFP 3 C00029 BC00029  +REFP EC00029
CALL JOB:SEARCH-R1-S13D
SET P033 P006
SFTON3D P033
SMOVL C00030 BC00030 V=166.7  +MOVJ EC00030
MOVL C00031 BC00031 V=1000.0  +MOVJ EC00031 VJ=100.00
'EndPath S3715
'Path S3716
SFTOF3D
MOVJ C00032 BC00032 VJ=100.00  +MOVJ EC00032 VJ=100.00
MOVL C00033 BC00033 V=800.0  +MOVJ EC00033 VJ=100.00
SMOVL C00034 BC00034 V=166.7  +MOVJ EC00034
SREFP 3 C00035 BC00035  +REFP EC00035
CALL JOB:SEARCH-R1-S13D
SET P032 P006
SFTON3D P032
SMOVL C00036 BC00036 V=166.7  +MOVJ EC00036
SMOVL C00037 BC00037 V=166.7  +MOVJ EC00037
SREFP 3 C00038 BC00038  +REFP EC00038
CALL JOB:SEARCH-R1-S13D
SET P032 P006
SFTON3D P032
SMOVL C00039 BC00039 V=166.7  +MOVJ EC00039
SMOVL C00040 BC00040 V=166.7  +MOVJ EC00040
SREFP 3 C00041 BC00041  +REFP EC00041
CALL JOB:SEARCH-R1-S13D
SET P032 P006
SFTON3D P032
SMOVL C00042 BC00042 V=166.7  +MOVJ EC00042
MOVL C00043 BC00043 V=1000.0  +MOVJ EC00043 VJ=100.00
'EndPath S3716
MOVJ C00044 BC00044 VJ=100.00  +MOVJ EC00044 VJ=100.00
'Path S3717
SFTOF3D
MOVJ C00045 BC00045 VJ=100.00  +MOVJ EC00045 VJ=100.00
MOVJ C00046 BC00046 VJ=100.00  +MOVJ EC00046 VJ=100.00
'Path S4334
SFTOF3D
MOVJ C00047 BC00047 VJ=100.00  +MOVJ EC00047 VJ=100.00
MOVL C00048 BC00048 V=800.0  +MOVJ EC00048 VJ=100.00
SMOVL C00049 BC00049 V=166.7  +MOVJ EC00049
SREFP 3 C00050 BC00050  +REFP EC00050
CALL JOB:SEARCH-R1-S13D
SET P029 P006
SFTON3D P029
SMOVL C00051 BC00051 V=166.7  +MOVJ EC00051
SMOVL C00052 BC00052 V=166.7  +MOVJ EC00052
SREFP 3 C00053 BC00053  +REFP EC00053
CALL JOB:SEARCH-R1-S13D
SET P029 P006
SFTON3D P029
SMOVL C00054 BC00054 V=166.7  +MOVJ EC00054
MOVL C00055 BC00055 V=800.0  +MOVJ EC00055 VJ=100.00
MOVL C00056 BC00056 V=1000.0  +MOVJ EC00056 VJ=100.00
SFTOF3D
SMOVL C00057 BC00057 V=166.7  +MOVJ EC00057
SREFP 3 C00058 BC00058  +REFP EC00058
CALL JOB:SEARCH-R1-S13D
SET P060 P006
SFTON3D P060
SMOVL C00059 BC00059 V=166.7  +MOVJ EC00059
SREFP 3 C00060 BC00060  +REFP EC00060
CALL JOB:SEARCH-R1-S13D
SET P060 P006
SFTON3D P060
SMOVL C00061 BC00061 V=166.7  +MOVJ EC00061
SMOVL C00062 BC00062 V=166.7  +MOVJ EC00062
SMOVL C00063 BC00063 V=166.7  +MOVJ EC00063
SREFP 3 C00064 BC00064  +REFP EC00064
CALL JOB:SEARCH-R1-S13D
SET P060 P006
SFTON3D P060
SMOVL C00065 BC00065 V=166.7  +MOVJ EC00065
SFTOF3D
'POPAWIC SERCH
SMOVL C00066 BC00066 V=166.7  +MOVJ EC00066
SMOVL C00067 BC00067 V=250.0  +MOVJ EC00067
SMOVL C00068 BC00068 V=250.0  +MOVJ EC00068
SREFP 3 C00069 BC00069  +REFP EC00069
CALL JOB:SEARCH-R1-S13D
SET P061 P006
SFTON3D P061
SMOVL C00070 BC00070 V=166.7  +MOVJ EC00070
SREFP 3 C00071 BC00071  +REFP EC00071
CALL JOB:SEARCH-R1-S13D
SET P061 P006
SFTON3D P061
SMOVL C00072 BC00072 V=166.7  +MOVJ EC00072
SMOVL C00073 BC00073 V=333.3  +MOVJ EC00073
SMOVL C00074 BC00074 V=250.0  +MOVJ EC00074
SREFP 3 C00075 BC00075  +REFP EC00075
CALL JOB:SEARCH-R1-S13D
SET P061 P006
SFTON3D P061
SMOVL C00076 BC00076 V=333.3  +MOVJ EC00076
SFTOF3D
'EndPath S4334
MOVJ C00077 BC00077 VJ=100.00  +MOVJ EC00077 VJ=100.00
MOVJ C00078 BC00078 VJ=100.00  +MOVJ EC00078 VJ=100.00
MOVJ C00079 BC00079 VJ=100.00  +MOVJ EC00079 VJ=100.00
SMOVL C00080 BC00080 V=150.0  +MOVJ EC00080
SREFP 3 C00081 BC00081  +REFP EC00081
CALL JOB:SEARCH-R1-S13D
SET P099 P006
SFTON3D P099
SMOVL C00082 BC00082 V=166.7  +MOVJ EC00082
SMOVL C00083 BC00083 V=250.0  +MOVJ EC00083
SMOVL C00084 BC00084 V=166.7  +MOVJ EC00084
SREFP 3 C00085 BC00085  +REFP EC00085
CALL JOB:SEARCH-R1-S13D
SET P099 P006
SFTON3D P099
SMOVL C00086 BC00086 V=250.0  +MOVJ EC00086
MOVJ C00087 BC00087 VJ=100.00  +MOVJ EC00087 VJ=100.00
MOVJ C00088 BC00088 VJ=100.00  +MOVJ EC00088 VJ=100.00
'Path S4335
SFTOF3D
MOVJ C00089 BC00089 VJ=100.00  +MOVJ EC00089 VJ=100.00
MOVL C00090 BC00090 V=800.0  +MOVJ EC00090 VJ=100.00
SMOVL C00091 BC00091 V=166.7  +MOVJ EC00091
SREFP 3 C00092 BC00092  +REFP EC00092
CALL JOB:SEARCH-R1-S13D
SET P028 P006
SFTON3D P028
SMOVL C00093 BC00093 V=166.7  +MOVJ EC00093
SMOVL C00094 BC00094 V=166.7  +MOVJ EC00094
SREFP 3 C00095 BC00095  +REFP EC00095
CALL JOB:SEARCH-R1-S13D
SET P028 P006
SFTON3D P028
SMOVL C00096 BC00096 V=166.7  +MOVJ EC00096
MOVL C00097 BC00097 V=800.0  +MOVJ EC00097 VJ=100.00
MOVL C00098 BC00098 V=1000.0  +MOVJ EC00098 VJ=100.00
'EndPath S4335
'Path S4336
SFTOF3D
MOVJ C00099 BC00099 VJ=100.00  +MOVJ EC00099 VJ=100.00
MOVL C00100 BC00100 V=800.0  +MOVJ EC00100 VJ=100.00
SMOVL C00101 BC00101 V=166.7  +MOVJ EC00101
SREFP 3 C00102 BC00102  +REFP EC00102
CALL JOB:SEARCH-R1-S13D
SET P027 P006
SFTON3D P027
SMOVL C00103 BC00103 V=166.7  +MOVJ EC00103
SMOVL C00104 BC00104 V=166.7  +MOVJ EC00104
SREFP 3 C00105 BC00105  +REFP EC00105
CALL JOB:SEARCH-R1-S13D
SET P027 P006
SFTON3D P027
SMOVL C00106 BC00106 V=166.7  +MOVJ EC00106
SMOVL C00107 BC00107 V=250.0  +MOVJ EC00107
SMOVL C00108 BC00108 V=166.7  +MOVJ EC00108
SREFP 3 C00109 BC00109  +REFP EC00109
CALL JOB:SEARCH-R1-S13D
SET P027 P006
SFTON3D P027
SMOVL C00110 BC00110 V=166.7  +MOVJ EC00110
SFTOF3D
MOVL C00111 BC00111 V=800.0  +MOVJ EC00111 VJ=100.00
MOVL C00112 BC00112 V=1000.0  +MOVJ EC00112 VJ=100.00
'EndPath S4336
'Up
MOVJ C00113 BC00113 VJ=100.00  +MOVJ EC00113 VJ=100.00
MOVJ C00114 BC00114 VJ=100.00  +MOVJ EC00114 VJ=100.00
MOVJ C00115 BC00115 VJ=100.00  +MOVJ EC00115 VJ=100.00
'Path S3719
SFTOF3D
MOVJ C00116 BC00116 VJ=100.00  +MOVJ EC00116 VJ=100.00
MOVL C00117 BC00117 V=800.0  +MOVJ EC00117 VJ=100.00
SMOVL C00118 BC00118 V=166.7  +MOVJ EC00118
SREFP 3 C00119 BC00119  +REFP EC00119
CALL JOB:SEARCH-R1-S13D
SET P026 P006
SFTON3D P026
SMOVL C00120 BC00120 V=166.7  +MOVJ EC00120
SREFP 3 C00121 BC00121  +REFP EC00121
CALL JOB:SEARCH-R1-S13D
SET P026 P006
SFTON3D P026
SMOVL C00122 BC00122 V=166.7  +MOVJ EC00122
MOVL C00123 BC00123 V=1000.0  +MOVJ EC00123 VJ=100.00
'EndPath S3719
'Path S4337
SFTOF3D
MOVJ C00124 BC00124 VJ=100.00  +MOVJ EC00124 VJ=100.00
MOVL C00125 BC00125 V=800.0  +MOVJ EC00125 VJ=100.00
SMOVL C00126 BC00126 V=166.7  +MOVJ EC00126
SREFP 3 C00127 BC00127  +REFP EC00127
CALL JOB:SEARCH-R1-S13D
SET P025 P006
SFTON3D P025
SMOVL C00128 BC00128 V=166.7  +MOVJ EC00128
SREFP 3 C00129 BC00129  +REFP EC00129
CALL JOB:SEARCH-R1-S13D
SET P025 P006
SFTON3D P025
SMOVL C00130 BC00130 V=166.7  +MOVJ EC00130
SMOVL C00131 BC00131 V=166.7  +MOVJ EC00131
SREFP 3 C00132 BC00132  +REFP EC00132
CALL JOB:SEARCH-R1-S13D
SET P025 P006
SFTON3D P025
SMOVL C00133 BC00133 V=166.7  +MOVJ EC00133
MOVL C00134 BC00134 V=1000.0  +MOVJ EC00134 VJ=100.00
'EndPath S4337
'Path S4338
SFTOF3D
MOVJ C00135 BC00135 VJ=100.00  +MOVJ EC00135 VJ=100.00
MOVL C00136 BC00136 V=800.0  +MOVJ EC00136 VJ=100.00
SMOVL C00137 BC00137 V=166.7  +MOVJ EC00137
SREFP 3 C00138 BC00138  +REFP EC00138
CALL JOB:SEARCH-R1-S13D
SET P024 P006
SFTON3D P024
SMOVL C00139 BC00139 V=166.7  +MOVJ EC00139
SREFP 3 C00140 BC00140  +REFP EC00140
CALL JOB:SEARCH-R1-S13D
SET P024 P006
SFTON3D P024
SMOVL C00141 BC00141 V=166.7  +MOVJ EC00141
SMOVL C00142 BC00142 V=166.7  +MOVJ EC00142
SREFP 3 C00143 BC00143  +REFP EC00143
CALL JOB:SEARCH-R1-S13D
SET P024 P006
SFTON3D P024
SMOVL C00144 BC00144 V=166.7  +MOVJ EC00144
MOVL C00145 BC00145 V=1000.0  +MOVJ EC00145 VJ=100.00
'EndPath S4338
'Path S3720
SFTOF3D
MOVJ C00146 BC00146 VJ=100.00  +MOVJ EC00146 VJ=100.00
MOVL C00147 BC00147 V=800.0  +MOVJ EC00147 VJ=100.00
SMOVL C00148 BC00148 V=166.7  +MOVJ EC00148
SREFP 3 C00149 BC00149  +REFP EC00149
CALL JOB:SEARCH-R1-S13D
SET P023 P006
SFTON3D P023
SMOVL C00150 BC00150 V=166.7  +MOVJ EC00150
SREFP 3 C00151 BC00151  +REFP EC00151
CALL JOB:SEARCH-R1-S13D
SET P023 P006
SFTON3D P023
SMOVL C00152 BC00152 V=166.7  +MOVJ EC00152
SMOVL C00153 BC00153 V=166.7  +MOVJ EC00153
SREFP 3 C00154 BC00154  +REFP EC00154
CALL JOB:SEARCH-R1-S13D
SET P023 P006
SFTON3D P023
SMOVL C00155 BC00155 V=166.7  +MOVJ EC00155
MOVL C00156 BC00156 V=1000.0  +MOVJ EC00156 VJ=100.00
'EndPath S3720
'Path S4726
SFTOF3D
MOVJ C00157 BC00157 VJ=100.00  +MOVJ EC00157 VJ=100.00
MOVL C00158 BC00158 V=800.0  +MOVJ EC00158 VJ=100.00
SMOVL C00159 BC00159 V=166.7  +MOVJ EC00159
SREFP 3 C00160 BC00160  +REFP EC00160
CALL JOB:SEARCH-R1-S13D
SET P063 P006
SFTON3D P063
SMOVL C00161 BC00161 V=166.7  +MOVJ EC00161
SMOVL C00162 BC00162 V=166.7  +MOVJ EC00162
SREFP 3 C00163 BC00163  +REFP EC00163
CALL JOB:SEARCH-R1-S13D
SET P063 P006
SFTON3D P063
SMOVL C00164 BC00164 V=166.7  +MOVJ EC00164
SMOVL C00165 BC00165 V=166.7  +MOVJ EC00165
SREFP 3 C00166 BC00166  +REFP EC00166
CALL JOB:SEARCH-R1-S13D
SET P063 P006
SFTON3D P063
SMOVL C00167 BC00167 V=166.7  +MOVJ EC00167
MOVL C00168 BC00168 V=1000.0  +MOVJ EC00168 VJ=100.00
'EndPath S4726
'Path S3721
SFTOF3D
MOVJ C00169 BC00169 VJ=100.00  +MOVJ EC00169 VJ=100.00
MOVL C00170 BC00170 V=800.0  +MOVJ EC00170 VJ=100.00
SMOVL C00171 BC00171 V=166.7  +MOVJ EC00171
SREFP 3 C00172 BC00172  +REFP EC00172
CALL JOB:SEARCH-R1-S13D
SET P022 P006
SFTON3D P022
SMOVL C00173 BC00173 V=166.7  +MOVJ EC00173
SREFP 3 C00174 BC00174  +REFP EC00174
CALL JOB:SEARCH-R1-S13D
SET P022 P006
SFTON3D P022
SMOVL C00175 BC00175 V=166.7  +MOVJ EC00175
SREFP 3 C00176 BC00176  +REFP EC00176
CALL JOB:SEARCH-R1-S13D
SET P022 P006
SFTON3D P022
SMOVL C00177 BC00177 V=166.7  +MOVJ EC00177
MOVL C00178 BC00178 V=1000.0  +MOVJ EC00178 VJ=100.00
'EndPath S3721
'Path S3722
SFTOF3D
MOVJ C00179 BC00179 VJ=100.00  +MOVJ EC00179 VJ=100.00
MOVL C00180 BC00180 V=800.0  +MOVJ EC00180 VJ=100.00
SMOVL C00181 BC00181 V=166.7  +MOVJ EC00181
SREFP 3 C00182 BC00182  +REFP EC00182
CALL JOB:SEARCH-R1-S13D
SET P021 P006
SFTON3D P021
SMOVL C00183 BC00183 V=166.7  +MOVJ EC00183
SREFP 3 C00184 BC00184  +REFP EC00184
CALL JOB:SEARCH-R1-S13D
SET P021 P006
SFTON3D P021
SMOVL C00185 BC00185 V=166.7  +MOVJ EC00185
SMOVL C00186 BC00186 V=166.7  +MOVJ EC00186
SREFP 3 C00187 BC00187  +REFP EC00187
CALL JOB:SEARCH-R1-S13D
SET P021 P006
SFTON3D P021
SMOVL C00188 BC00188 V=166.7  +MOVJ EC00188
MOVL C00189 BC00189 V=1000.0  +MOVJ EC00189 VJ=100.00
'EndPath S3722
MOVJ C00190 BC00190 VJ=100.00  +MOVJ EC00190 VJ=100.00
MOVJ C00191 BC00191 VJ=100.00  +MOVJ EC00191 VJ=100.00
'Path W4727
SFTOF3D
SFTON3D P024
MOVJ C00192 BC00192 VJ=100.00  +MOVJ EC00192 VJ=100.00
SMOVL C00193 BC00193 V=800.0  +MOVJ EC00193
SMOVL C00194 BC00194 V=150.0 PL=0  +MOVJ EC00194
MACRO1 MJ#(0) ARGF14
ARCON
SMOVL C00195 BC00195 V=10.0  +MOVJ EC00195
SMOVL C00196 BC00196 V=10.0  +MOVJ EC00196
ARCOF
SMOVL C00197 BC00197 V=800.0  +MOVJ EC00197
SMOVL C00198 BC00198 V=1000.0  +MOVJ EC00198
SFTOF3D
'EndPath W4727
MOVJ C00199 BC00199 VJ=100.00  +MOVJ EC00199 VJ=100.00
'Path W4728
SFTOF3D
SFTON3D P063
MOVJ C00200 BC00200 VJ=100.00  +MOVJ EC00200 VJ=100.00
SMOVL C00201 BC00201 V=800.0  +MOVJ EC00201
SMOVL C00202 BC00202 V=150.0 PL=0  +MOVJ EC00202
ARCON
SMOVL C00203 BC00203 V=10.0  +MOVJ EC00203
SMOVL C00204 BC00204 V=10.0  +MOVJ EC00204
ARCOF
SMOVL C00205 BC00205 V=800.0  +MOVJ EC00205
SMOVL C00206 BC00206 V=1000.0  +MOVJ EC00206
SFTOF3D
'EndPath W4728
'Path W3723
SFTOF3D
SFTON3D P021
MOVJ C00207 BC00207 VJ=100.00  +MOVJ EC00207 VJ=100.00
SMOVL C00208 BC00208 V=800.0  +MOVJ EC00208
SMOVL C00209 BC00209 V=166.7 PL=0  +MOVJ EC00209
MACRO1 MJ#(0) ARGF9
ARCON
SMOVL C00210 BC00210 V=10.0  +MOVJ EC00210
SFTON3D P022
SMOVL C00211 BC00211 V=10.0  +MOVJ EC00211
SMOVL C00212 BC00212 V=10.0  +MOVJ EC00212
ARCOF
SMOVL C00213 BC00213 V=800.0  +MOVJ EC00213
SMOVL C00214 BC00214 V=1000.0  +MOVJ EC00214
SFTOF3D
'EndPath W3723
MOVJ C00215 BC00215 VJ=100.00  +MOVJ EC00215 VJ=100.00
'Path W3724
SFTOF3D
SFTON3D P022
MOVJ C00216 BC00216 VJ=100.00  +MOVJ EC00216 VJ=100.00
SMOVL C00217 BC00217 V=800.0  +MOVJ EC00217
SMOVL C00218 BC00218 V=166.7 PL=0  +MOVJ EC00218
ARCON
SMOVL C00219 BC00219 V=10.0  +MOVJ EC00219
ARCOF
SMOVL C00220 BC00220 V=800.0  +MOVJ EC00220
SMOVL C00221 BC00221 V=1000.0  +MOVJ EC00221
SFTOF3D
'EndPath W3724
'Path W3725
SFTOF3D
SFTON3D P023
MOVJ C00222 BC00222 VJ=100.00  +MOVJ EC00222 VJ=100.00
SMOVL C00223 BC00223 V=800.0  +MOVJ EC00223
SMOVL C00224 BC00224 V=166.7 PL=0  +MOVJ EC00224
ARCON
SWVON WEV#(60)
SMOVL C00225 BC00225 V=7.5  +MOVJ EC00225
SFTON3D P024
SMOVL C00226 BC00226 V=7.5  +MOVJ EC00226
SMOVL C00227 BC00227 V=7.5  +MOVJ EC00227
ARCOF
SWVOF
SMOVL C00228 BC00228 V=800.0  +MOVJ EC00228
SMOVL C00229 BC00229 V=1000.0  +MOVJ EC00229
SFTOF3D
'EndPath W3725
'Path W3726
SFTOF3D
SFTON3D P025
MOVJ C00230 BC00230 VJ=100.00  +MOVJ EC00230 VJ=100.00
SMOVL C00231 BC00231 V=800.0  +MOVJ EC00231
SMOVL C00232 BC00232 V=166.7 PL=0  +MOVJ EC00232
ARCON
SMOVL C00233 BC00233 V=10.0  +MOVJ EC00233
SFTON3D P026
SMOVL C00234 BC00234 V=10.0  +MOVJ EC00234
SMOVL C00235 BC00235 V=10.0  +MOVJ EC00235
SMOVL C00236 BC00236 V=10.0  +MOVJ EC00236
ARCOF
SFTOF3D
SMOVL C00237 BC00237 V=800.0  +MOVJ EC00237
SMOVL C00238 BC00238 V=1000.0  +MOVJ EC00238
SFTOF3D
'EndPath W3726
'Down
MOVJ C00239 BC00239 VJ=100.00  +MOVJ EC00239 VJ=100.00
MOVJ C00240 BC00240 VJ=100.00  +MOVJ EC00240 VJ=100.00
MOVJ C00241 BC00241 VJ=100.00  +MOVJ EC00241 VJ=100.00
'Path W3727
SFTOF3D
SFTON3D P030
MOVJ C00242 BC00242 VJ=100.00  +MOVJ EC00242 VJ=100.00
MOVJ C00243 BC00243 VJ=100.00  +MOVJ EC00243 VJ=100.00
'Path W3729
SFTOF3D
SFTON3D P033
MOVJ C00244 BC00244 VJ=100.00  +MOVJ EC00244 VJ=100.00
SMOVL C00245 BC00245 V=800.0  +MOVJ EC00245
SMOVL C00246 BC00246 V=166.7 PL=0  +MOVJ EC00246
MACRO1 MJ#(0) ARGF14
ARCON
SMOVL C00247 BC00247 V=10.0  +MOVJ EC00247
ARCOF
SFTOF3D
SMOVL C00248 BC00248 V=800.0  +MOVJ EC00248
SMOVL C00249 BC00249 V=250.0  +MOVJ EC00249
SFTON3D P033
SMOVL C00250 BC00250 V=133.3  +MOVJ EC00250
ARCON
SMOVL C00251 BC00251 V=13.3  +MOVJ EC00251
ARCOF
SMOVL C00252 BC00252 V=166.7  +MOVJ EC00252
SMOVL C00253 BC00253 V=166.7  +MOVJ EC00253
SMOVL C00254 BC00254 V=166.7  +MOVJ EC00254
ARCON
SMOVL C00255 BC00255 V=13.3  +MOVJ EC00255
SMOVL C00256 BC00256 V=13.3  +MOVJ EC00256
ARCOF
SMOVL C00257 BC00257 V=166.7  +MOVJ EC00257
SMOVL C00258 BC00258 V=1000.0  +MOVJ EC00258
SFTOF3D
'EndPath W3729
'Path W3730
SFTOF3D
SFTON3D P032
MOVJ C00259 BC00259 VJ=100.00  +MOVJ EC00259 VJ=100.00
SMOVL C00260 BC00260 V=800.0  +MOVJ EC00260
SMOVL C00261 BC00261 V=166.7 PL=0  +MOVJ EC00261
ARCON
SMOVL C00262 BC00262 V=10.0  +MOVJ EC00262
SMOVL C00263 BC00263 V=11.7  +MOVJ EC00263
SMOVL C00264 BC00264 V=11.7  +MOVJ EC00264
ARCOF
SMOVL C00265 BC00265 V=166.7  +MOVJ EC00265
SMOVL C00266 BC00266 V=166.7  +MOVJ EC00266
MACRO1 MJ#(0) ARGF6
SMOVL C00267 BC00267 V=166.7  +MOVJ EC00267
ARCON
SMOVL C00268 BC00268 V=10.0  +MOVJ EC00268
ARCOF
SMOVL C00269 BC00269 V=166.7  +MOVJ EC00269
SMOVL C00270 BC00270 V=1000.0  +MOVJ EC00270
SFTOF3D
MOVJ C00271 BC00271 VJ=100.00  +MOVJ EC00271 VJ=100.00
'EndPath W3730
'Path W3731
SFTOF3D
SFTON3D P032
SFTOF3D
'EndPath W3731
'Path W4471
SFTOF3D
SFTON3D P027
MOVJ C00272 BC00272 VJ=100.00  +MOVJ EC00272 VJ=100.00
SMOVL C00273 BC00273 V=800.0  +MOVJ EC00273
SMOVL C00274 BC00274 V=150.0 PL=0  +MOVJ EC00274
MACRO1 MJ#(0) ARGF9
ARCON
SMOVL C00275 BC00275 V=10.8  +MOVJ EC00275
SMOVL C00276 BC00276 V=10.8  +MOVJ EC00276
ARCOF
SMOVL C00277 BC00277 V=800.0  +MOVJ EC00277
SMOVL C00278 BC00278 V=83.3  +MOVJ EC00278
ARCON
SMOVL C00279 BC00279 V=10.0  +MOVJ EC00279
ARCOF
SMOVL C00280 BC00280 V=250.0  +MOVJ EC00280
SMOVL C00281 BC00281 V=1000.0  +MOVJ EC00281
SFTOF3D
'EndPath W4471
MOVJ C00282 BC00282 VJ=100.00  +MOVJ EC00282 VJ=100.00
MOVJ C00283 BC00283 VJ=100.00  +MOVJ EC00283 VJ=100.00
'Path W4472
SFTOF3D
SFTON3D P027
MOVJ C00284 BC00284 VJ=100.00  +MOVJ EC00284 VJ=100.00
SMOVL C00285 BC00285 V=800.0  +MOVJ EC00285
SMOVL C00286 BC00286 V=150.0 PL=0  +MOVJ EC00286
ARCON
SMOVL C00287 BC00287 V=10.8  +MOVJ EC00287
ARCOF
SMOVL C00288 BC00288 V=800.0  +MOVJ EC00288
SMOVL C00289 BC00289 V=1000.0  +MOVJ EC00289
SFTOF3D
'EndPath W4472
'Path W4473
SFTOF3D
SFTON3D P028
MOVJ C00290 BC00290 VJ=100.00  +MOVJ EC00290 VJ=100.00
SMOVL C00291 BC00291 V=800.0  +MOVJ EC00291
SMOVL C00292 BC00292 V=150.0 PL=0  +MOVJ EC00292
ARCON
SMOVL C00293 BC00293 V=10.8  +MOVJ EC00293
ARCOF
SMOVL C00294 BC00294 V=800.0  +MOVJ EC00294
SMOVL C00295 BC00295 V=1000.0  +MOVJ EC00295
SFTOF3D
'EndPath W4473
'Path W4474
SFTOF3D
SFTON3D P028
MOVJ C00296 BC00296 VJ=100.00  +MOVJ EC00296 VJ=100.00
SMOVL C00297 BC00297 V=800.0  +MOVJ EC00297
SMOVL C00298 BC00298 V=150.0 PL=0  +MOVJ EC00298
ARCON
SMOVL C00299 BC00299 V=10.8  +MOVJ EC00299
SMOVL C00300 BC00300 V=10.8  +MOVJ EC00300
ARCOF
SMOVL C00301 BC00301 V=800.0  +MOVJ EC00301
SMOVL C00302 BC00302 V=1000.0  +MOVJ EC00302
SFTOF3D
'EndPath W4474
MOVJ C00303 BC00303 VJ=100.00  +MOVJ EC00303 VJ=100.00
MOVJ C00304 BC00304 VJ=100.00  +MOVJ EC00304 VJ=100.00
'Path W4477
SFTOF3D
SFTON3D P029
MOVJ C00305 BC00305 VJ=100.00  +MOVJ EC00305 VJ=100.00
SMOVL C00306 BC00306 V=800.0  +MOVJ EC00306
SMOVL C00307 BC00307 V=150.0 PL=0  +MOVJ EC00307
ARCON
SMOVL C00308 BC00308 V=10.8  +MOVJ EC00308
ARCOF
SMOVL C00309 BC00309 V=800.0  +MOVJ EC00309
SMOVL C00310 BC00310 V=1000.0  +MOVJ EC00310
SFTOF3D
'EndPath W4477
MOVJ C00311 BC00311 VJ=100.00  +MOVJ EC00311 VJ=100.00
MOVJ C00312 BC00312 VJ=100.00  +MOVJ EC00312 VJ=100.00
'Path W4478
SFTOF3D
SFTON3D P029
MOVJ C00313 BC00313 VJ=100.00  +MOVJ EC00313 VJ=100.00
SMOVL C00314 BC00314 V=800.0  +MOVJ EC00314
SMOVL C00315 BC00315 V=150.0 PL=0  +MOVJ EC00315
ARCON
SMOVL C00316 BC00316 V=10.8  +MOVJ EC00316
ARCOF
SMOVL C00317 BC00317 V=800.0  +MOVJ EC00317
SMOVL C00318 BC00318 V=1000.0  +MOVJ EC00318
SFTOF3D
'EndPath W4478
MOVJ C00319 BC00319 VJ=100.00  +MOVJ EC00319 VJ=100.00
MOVJ C00320 BC00320 VJ=100.00  +MOVJ EC00320 VJ=100.00
SFTON3D P060
MACRO1 MJ#(0) ARGF14
SMOVL C00321 BC00321 V=166.7  +MOVJ EC00321
ARCON
SMOVL C00322 BC00322 V=11.7  +MOVJ EC00322
ARCOF
SMOVL C00323 BC00323 V=133.3  +MOVJ EC00323
SMOVL C00324 BC00324 V=133.3  +MOVJ EC00324
SMOVL C00325 BC00325 V=133.3  +MOVJ EC00325
ARCON
SMOVL C00326 BC00326 V=10.8  +MOVJ EC00326
ARCOF
SMOVL C00327 BC00327 V=333.3  +MOVJ EC00327
MOVJ C00328 BC00328 VJ=100.00  +MOVJ EC00328 VJ=100.00
SFTOF3D
MOVJ C00329 BC00329 VJ=100.00  +MOVJ EC00329 VJ=100.00
MOVJ C00330 BC00330 VJ=100.00  +MOVJ EC00330 VJ=100.00
SFTON3D P061
SMOVL C00331 BC00331 V=133.3  +MOVJ EC00331
ARCON
SMOVL C00332 BC00332 V=11.7  +MOVJ EC00332
ARCOF
SMOVL C00333 BC00333 V=166.7  +MOVJ EC00333
MOVJ C00334 BC00334 VJ=100.00  +MOVJ EC00334 VJ=100.00
MOVJ C00335 BC00335 VJ=100.00  +MOVJ EC00335 VJ=100.00
MOVJ C00336 BC00336 VJ=100.00  +MOVJ EC00336 VJ=100.00
SMOVL C00337 BC00337 V=166.7  +MOVJ EC00337
ARCON
SMOVL C00338 BC00338 V=11.7  +MOVJ EC00338
ARCOF
SMOVL C00339 BC00339 V=133.3  +MOVJ EC00339
COMM SMOVL C00340 BC00340 V=166.7  +MOVJ EC00340
COMM ARCON
COMM SMOVL C00341 BC00341 V=6.7  +MOVJ EC00341
COMM ARCOF
COMM SMOVL C00342 BC00342 V=83.3  +MOVJ EC00342
COMM SMOVL C00343 BC00343 V=166.7  +MOVJ EC00343
COMM SMOVL C00344 BC00344 V=83.3  +MOVJ EC00344
COMM ARCON
COMM SMOVL C00345 BC00345 V=6.7  +MOVJ EC00345
COMM ARCOF
COMM SMOVL C00346 BC00346 V=166.7  +MOVJ EC00346
SFTOF3D
SMOVL C00347 BC00347 V=800.0  +MOVJ EC00347
MOVJ C00348 BC00348 VJ=100.00  +MOVJ EC00348 VJ=100.00
MOVJ C00349 BC00349 VJ=100.00  +MOVJ EC00349 VJ=100.00
MOVJ C00350 BC00350 VJ=100.00  +MOVJ EC00350 VJ=100.00
MOVJ C00351 BC00351 VJ=100.00  +MOVJ EC00351 VJ=100.00
SFTON3D P060
SMOVL C00352 BC00352 V=133.3  +MOVJ EC00352
ARCON
SMOVL C00353 BC00353 V=11.7  +MOVJ EC00353
ARCOF
SMOVL C00354 BC00354 V=250.0  +MOVJ EC00354
SFTOF3D
MOVJ C00355 BC00355 VJ=100.00  +MOVJ EC00355 VJ=100.00
MOVJ C00356 BC00356 VJ=100.00  +MOVJ EC00356 VJ=100.00
MOVJ C00357 BC00357 VJ=100.00  +MOVJ EC00357 VJ=100.00
MACRO1 MJ#(0) ARGF6
SFTON3D P027
SMOVL C00358 BC00358 V=133.3  +MOVJ EC00358
ARCON
SMOVL C00359 BC00359 V=15.0  +MOVJ EC00359
ARCOF
SFTOF3D
SMOVL C00360 BC00360 V=15.0  +MOVJ EC00360
SMOVL C00361 BC00361 V=15.0  +MOVJ EC00361
ARCOF
SMOVL C00362 BC00362 V=166.7  +MOVJ EC00362
SMOVL C00363 BC00363 V=666.7  +MOVJ EC00363
MOVJ C00364 BC00364 VJ=100.00  +MOVJ EC00364 VJ=100.00
MOVJ C00365 BC00365 VJ=100.00  +MOVJ EC00365 VJ=100.00
'Path W3732
SFTOF3D
SFTON3D P034
MOVJ C00366 BC00366 VJ=100.00  +MOVJ EC00366 VJ=100.00
MOVJ C00367 BC00367 VJ=100.00  +MOVJ EC00367 VJ=100.00
SMOVL C00368 BC00368 V=800.0  +MOVJ EC00368
SMOVL C00369 BC00369 V=150.0 PL=0  +MOVJ EC00369
MACRO1 MJ#(0) ARGF14
ARCON
SMOVL C00370 BC00370 V=11.7  +MOVJ EC00370
SMOVL C00371 BC00371 V=11.7  +MOVJ EC00371
ARCOF
SMOVL C00372 BC00372 V=800.0  +MOVJ EC00372
SMOVL C00373 BC00373 V=500.0  +MOVJ EC00373
COMM MOVJ C00374 BC00374 VJ=100.00  +MOVJ EC00374 VJ=100.00
COMM MOVJ C00375 BC00375 VJ=100.00  +MOVJ EC00375 VJ=100.00
COMM MOVJ C00376 BC00376 VJ=100.00  +MOVJ EC00376 VJ=100.00
SFTON3D P034
SMOVL C00377 BC00377 V=133.3  +MOVJ EC00377
ARCON
SMOVL C00378 BC00378 V=11.7  +MOVJ EC00378
SMOVL C00379 BC00379 V=11.7  +MOVJ EC00379
ARCOF
SMOVL C00380 BC00380 V=166.7  +MOVJ EC00380
SMOVL C00381 BC00381 V=166.7  +MOVJ EC00381
SMOVL C00382 BC00382 V=166.7  +MOVJ EC00382
ARCON
SMOVL C00383 BC00383 V=10.0  +MOVJ EC00383
ARCOF
SMOVL C00384 BC00384 V=133.3  +MOVJ EC00384
SFTOF3D
SMOVL C00385 BC00385 V=333.3  +MOVJ EC00385
MOVJ C00386 BC00386 VJ=100.00  +MOVJ EC00386 VJ=100.00
MOVJ C00387 BC00387 VJ=100.00  +MOVJ EC00387 VJ=100.00
MOVJ C00388 BC00388 VJ=100.00  +MOVJ EC00388 VJ=100.00
MOVJ C00389 BC00389 VJ=100.00  +MOVJ EC00389 VJ=100.00
SFTON3D P099
SMOVL C00390 BC00390 V=166.7  +MOVJ EC00390
ARCON
SMOVL C00391 BC00391 V=11.7  +MOVJ EC00391
ARCOF
SMOVL C00392 BC00392 V=250.0  +MOVJ EC00392
'EndPath W3732
MOVJ C00393 BC00393 VJ=100.00  +MOVJ EC00393 VJ=100.00
MOVJ C00394 BC00394 VJ=100.00  +MOVJ EC00394 VJ=100.00
MOVJ C00395 BC00395 VJ=100.00  +MOVJ EC00395 VJ=100.00
END
